PROGRAM MAIN
VAR
	// HMI Variables
	HMI_bRun 	: BOOL;
	HMI_nPT1	: INT;
	
	// state machine
	eSystemState		: E_SystemState;

	// function blocks
	fbProcessCalcs		: FB_ProcessCalcs;
	fbFaultMonitor 		: FB_FaultMonitor;
	fbHmi 				: FB_Hmi;
	fbPressureControl 	: FB_PressureControl;
	fbPurge 			: FB_Purge;
	fbSpaFlush			: FB_SpaFlush;
	fbStateMachine 		: FB_StateMachine;
	fbWaterFill 		: FB_WaterFill;
	fbOutputHandler		: FB_OutputHandler;
	
	// fbWaterFill
	reqSV4_FillVavle			: BOOL;
	bLS1_WaterCenter_Filtered	: BOOL;
	bLS3_WaterEmpty_Filtered	: BOOL;
	
	// fbPurge
	reqSV1_DrainValve			: BOOL;
	
	// fbPresureControl
	reqH1_Upstream				: BOOL;
	
END_VAR

//========================= FB CALLS =====================================

// SCALE INPUTS
fbProcessCalcs(eState := fbStateMachine.eState);

// FAULT CHECK
fbFaultMonitor(
	stProcess := fbProcessCalcs.stProcessValues,
	eState := fbStateMachine.eState,
	bPurgeActive := fbStateMachine.bPurgeEnable,
	bWaterFillActive := (fbWaterFill.eMode = E_WaterFillMode.RunningAutofill) 
						 OR (fbWaterFill.eMode = E_WaterFillMode.StartupFill),
	bDiffPressActive := fbStateMachine.bControlEnable,
	bDiffPressReached := fbPressureControl.bDiffPressReached,
	bTempControlActive := fbStateMachine.bControlEnable,
	bColdStart := fbStateMachine.bColdStart,
	bReadyReached := fbStateMachine.bReady,
	bSteamFlowing := fbStateMachine.bDeliveryEnable,
	bWaterEmptyFiltered := fbWaterFill.bEmptyFiltered,
	bWaterCenterFiltered := fbWaterFill.bCenterFiltered,
	bExternalHeaterOff := NOT fbHmi.bCmdExtHeaterOn,
	bHmiHeartbeatOk := NOT fbHmi.bHmiCommLoss
	);

//========================= HMI (publish + consume) =======================
// Run BEFORE the state machine so command pulses are latched this cycle.
// FB_Hmi publishes GVL_HMI.stStatus and clears consumed command bits.
fbHmi(
	eState      := fbStateMachine.eState,
    stProcess   := fbProcessCalcs.stProcessValues,
	stFaults	:= fbFaultMonitor.stFaults,
	bReady 		:= fbStateMachine.bReady
);
	  
//========================= STATE MACHINE =================================
// Consume the one-cycle HMI command pulses, then run the CASE.
IF fbHmi.bCmdSesOn THEN fbStateMachine.RequestStart(); END_IF
IF fbHmi.bCmdSesOff THEN fbStateMachine.RequestStop(); END_IF
IF fbHmi.bCmdEnterMaint THEN fbStateMachine.RequestMaintenance(); END_IF
IF fbHmi.bCmdExitMaint THEN fbStateMachine.RequestExitMaint(); END_IF
IF fbHmi.bCmdFaultReset THEN
    fbFaultMonitor.ResetAll();
    fbStateMachine.RequestFaultReset();
END_IF;

// Latch fault -> force state machine into Fault (only auto-clears via reset).
IF fbFaultMonitor.bAnyLatchingFault THEN
    fbStateMachine.RequestFault();
END_IF

fbStateMachine(
	stFaults := fbFaultMonitor.stFaults,
	stHmiSetpoints := GVL_HMI.stHmiSetpoints,
	stProcessValues := fbProcessCalcs.stProcessValues,
	bDeliveryCmd := fbHmi.bCmdDelivery,
	bFillComplete := fbWaterFill.bFillComplete,
	bPurgeComplete := fbPurge.bPurgeComplete,
	rSpaTemp := fbProcessCalcs.stProcessValues.rTc1Spa,
	bSpaFlushed := fbSpaFlush.bSpaFlushed,
	eState => eSystemState
);
				
//========================= SUBROUTINES =================================
// Subroutines only run only when the state machine enables them. In Maintenance,
// the enable flags follow the HMI control-loop override toggles.

fbWaterFill(
	eMode := fbStateMachine.eWaterFillMode,
	bCenterSwitch := GVL_IO.biLS1_WaterMidLevel,
	bEmptySwitch := GVL_IO.biLS3_WaterLowLevel,
	bAutofillEnable := fbHmi.bCmdAutofillEnable,
	bFillComplete => GVL_HMI.stHmiStatus.bFillComplete,
	bCenterFiltered => GVL_HMI.stHmiStatus.stProcess.bWaterFull,
	bEmptyFiltered => GVL_HMI.stHmiStatus.stProcess.bWaterEmpty
);

fbPurge(
	bEnable :=fbStateMachine.bPurgeEnable,
	rUpstreamPress := fbProcessCalcs.stProcessValues.rPt1Upstream,
	bEmptyFiltered := fbWaterFill.bEmptyFiltered,
	bPurgeTimeout => GVL_HMI.stHmiStatus.stFaults.bPurgeTimeout
);
		
fbPressureControl(
	bEnable := fbStateMachine.bControlEnable,          
	eState := fbStateMachine.eState,        
	bDpControlOff := fbHmi.bCmdSuspendDpLoop,
	bTempControlOff := fbHmi.bCmdSuspendTempLoop,
	bExtHeaterEnable := fbHmi.bCmdExtHeaterOn,
	stProcess := fbProcessCalcs.stProcessValues,
	stSetpoints := GVL_HMI.stHmiSetpoints ,
	bFlushed := fbSpaFlush.bSpaFlushed
);

fbSpaFlush(
	bEnable := fbStateMachine.bSpaFlushEnable,
	bReset := fbStateMachine.bSpaFlushReset,
	rUpstreamPress := fbProcessCalcs.stProcessValues.rPt1Upstream,
	rAtmPressure := fbProcessCalcs.stProcessValues.rAtmPressure
);
	




//========================= OUTPUT HANDLER ====================================
fbOutputHandler(
	eState := fbStateMachine.eState,
	bWaterFillValve := fbWaterFill.qFillValve,
	bPurgeValve := fbPurge.qDrainValve,
	bDeliveryPermit := GVL_HMI.stHmiCommand.bSteamDeliveryOn,
	bH1Upstream := fbPressureControl.qH1_UpstreamHeater,
	bH2Purifier := fbPressureControl.qH2_SpaHeater,
	bFmHeater := fbPressureControl.qH3_FlowmeterHeater,
	bExtHeater := fbPressureControl.qH4_ExternalHeater,
	arValveOverride := GVL_HMI.stHmiCommand.aValveCmd,
	stProcess := fbProcessCalcs.stProcessValues
);

END_PROGRAM

(* stored: Version 1.1.0.1, ProductVersion 3.1.4026.19
   POU MAIN: Id {f6813ce8-0276-401c-9fea-66add7e7619a}, SpecialFunc None *)
